{attribute 'GeneratedUsingTerminal: AT2020-0250-0023'}
{attribute addProperty BoxType "AT2020-0250-0023"}
{attribute addProperty Id "A_0073_AT2000_5250_0016_AT2000_5250AT2000_33A3DF1B80"}
{attribute addProperty CRC "765113308"}
{attribute addProperty Size "80"}
TYPE A_0061_AT2020_0250_0023_AT2020_0250_2D9AB3DC EXTENDS AT2020_A7FEA1CF :
STRUCT
	{attribute addProperty Name "A_0073_AT2000_5250_0016_AT2000_5250"}
	{attribute addProperty PreviousPort "A_0061(AT2020-0250-0023) (AT2020-0250) : B"}
	A_0073_AT2000_5250_0016_AT2000_5250 : AT2000_33A3DF1B;
END_STRUCT
END_TYPE
